INTERFACE I_SingleMover EXTENDS I_Base

PROPERTY Mover1 : I_XPlanarMover
GET
END_GET
SET
END_SET
END_PROPERTY

METHOD SetMovers : BOOL
VAR_INPUT
	M1, M2 : I_XPlanarMover := 0;
END_VAR
END_METHOD

END_INTERFACE

(* stored: Version 1.1.0.1, ProductVersion 3.1.4026.20
   Itf I_SingleMover: Id {1ff7bed2-7eeb-4f40-90af-1b1f3234dee7}
   Property Mover1: Id {0b42ec4e-a5ed-4204-8ae1-4ff8ccd293de}
   Get Get: Id {f1b6d725-f47d-43b3-b285-1d847e8cc654}
   Set Set: Id {ab6a5751-3527-4c8c-af92-80017b83d095}
   Method SetMovers: Id {ccce57ef-481f-4c2c-b85f-c00d05032561} *)
